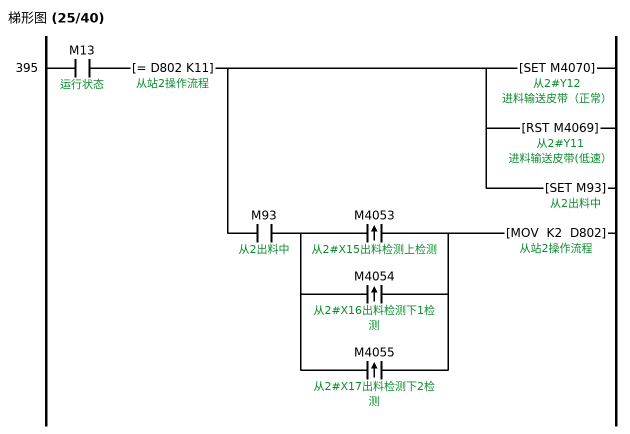
[picture p24: 梯形图 rows 395-395]
LD     M13	; 运行状态
AND=   D802 K11	; 从站2操作流程
SET    M4070	; 从2#Y12 进料输送皮带（正常）
RST    M4069	; 从2#Y11 进料输送皮带(低速）
SET    M93	; 从2出料中
AND    M93	; 从2出料中
LDP    M4053	; 从2#X15出料检测上检测
ORP    M4054	; 从2#X16出料检测下1检测
ORP    M4055	; 从2#X17出料检测下2检测
ANB
MOV    K2 D802	; 从站2操作流程

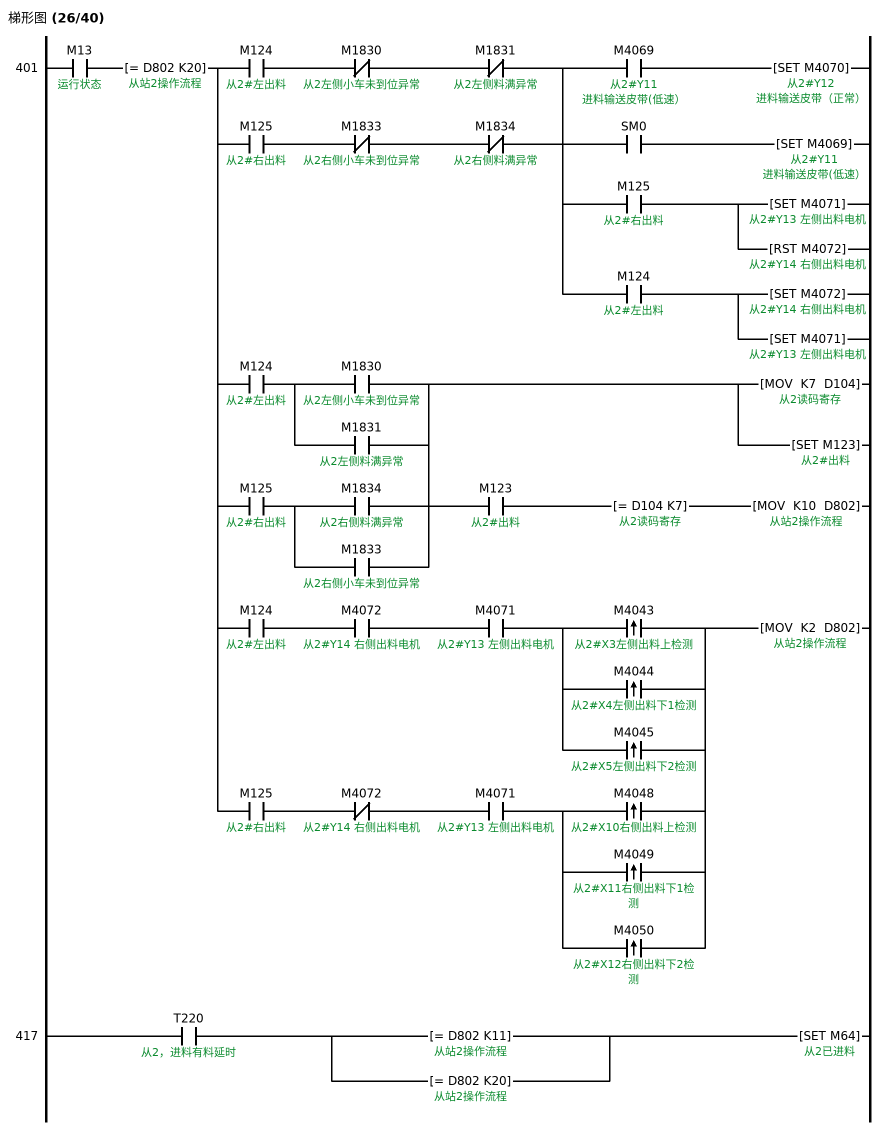
LD     M13	; 运行状态
AND=   D802 K20	; 从站2操作流程
MPS
LD     M124	; 从2#左出料
ANI    M1830	; 从2左侧小车未到位异常
ANI    M1831	; 从2左侧料满异常
LD     M125	; 从2#右出料
ANI    M1833	; 从2右侧小车未到位异常
ANI    M1834	; 从2右侧料满异常
ORB
ANB
MPS
AND    M4069	; 从2#Y11 进料输送皮带(低速）
SET    M4070	; 从2#Y12 进料输送皮带（正常）
MRD
AND    SM0
SET    M4069	; 从2#Y11 进料输送皮带(低速）
MRD
AND    M125	; 从2#右出料
SET    M4071	; 从2#Y13 左侧出料电机
RST    M4072	; 从2#Y14 右侧出料电机
MPP
AND    M124	; 从2#左出料
SET    M4072	; 从2#Y14 右侧出料电机
SET    M4071	; 从2#Y13 左侧出料电机
MRD
LD     M124	; 从2#左出料
LD     M1830	; 从2左侧小车未到位异常
OR     M1831	; 从2左侧料满异常
ANB
LD     M125	; 从2#右出料
LD     M1834	; 从2右侧料满异常
OR     M1833	; 从2右侧小车未到位异常
ANB
ORB
ANB
MOV    K7 D104	; 从2读码寄存
SET    M123	; 从2#出料
AND    M123	; 从2#出料
AND=   D104 K7	; 从2读码寄存
MOV    K10 D802	; 从站2操作流程
MPP
LD     M124	; 从2#左出料
AND    M4072	; 从2#Y14 右侧出料电机
AND    M4071	; 从2#Y13 左侧出料电机
LDP    M4043	; 从2#X3左侧出料上检测
ORP    M4044	; 从2#X4左侧出料下1检测
ORP    M4045	; 从2#X5左侧出料下2检测
ANB
LD     M125	; 从2#右出料
ANI    M4072	; 从2#Y14 右侧出料电机
AND    M4071	; 从2#Y13 左侧出料电机
LDP    M4048	; 从2#X10右侧出料上检测
ORP    M4049	; 从2#X11右侧出料下1检测
ORP    M4050	; 从2#X12右侧出料下2检测
ANB
ORB
ANB
MOV    K2 D802	; 从站2操作流程
LD     T220	; 从2，进料有料延时
LD=    D802 K11	; 从站2操作流程
OR=    D802 K20	; 从站2操作流程
ANB
SET    M64	; 从2已进料

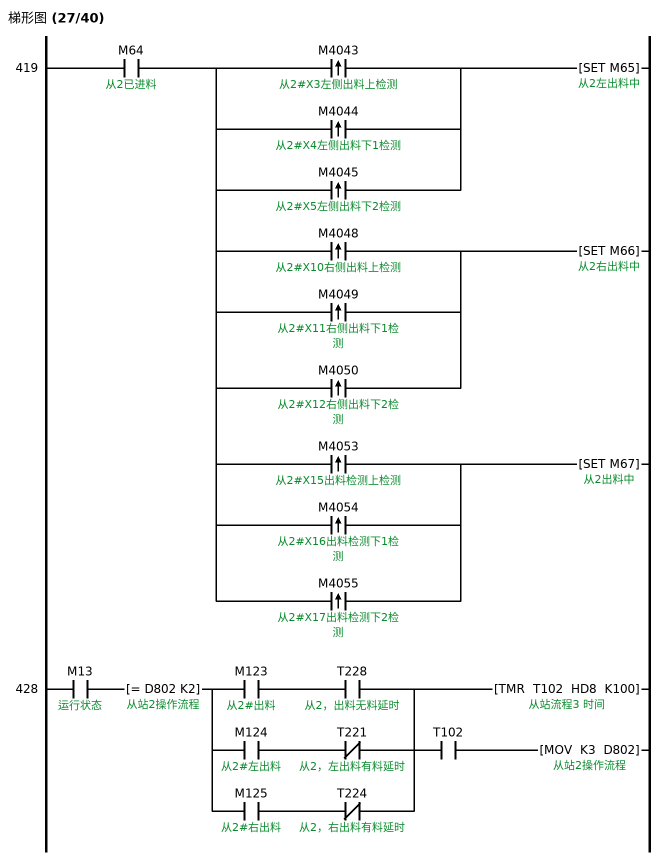
LD     M64	; 从2已进料
MPS
LDP    M4043	; 从2#X3左侧出料上检测
ORP    M4044	; 从2#X4左侧出料下1检测
ORP    M4045	; 从2#X5左侧出料下2检测
ANB
SET    M65	; 从2左出料中
MRD
LDP    M4048	; 从2#X10右侧出料上检测
ORP    M4049	; 从2#X11右侧出料下1检测
ORP    M4050	; 从2#X12右侧出料下2检测
ANB
SET    M66	; 从2右出料中
MPP
LDP    M4053	; 从2#X15出料检测上检测
ORP    M4054	; 从2#X16出料检测下1检测
ORP    M4055	; 从2#X17出料检测下2检测
ANB
SET    M67	; 从2出料中
LD     M13	; 运行状态
AND=   D802 K2	; 从站2操作流程
LD     M123	; 从2#出料
AND    T228	; 从2，出料无料延时
LD     M124	; 从2#左出料
ANI    T221	; 从2，左出料有料延时
ORB
LD     M125	; 从2#右出料
ANI    T224	; 从2，右出料有料延时
ORB
ANB
TMR    T102 HD8 K100	; 从站流程3 时间
AND    T102
MOV    K3 D802	; 从站2操作流程

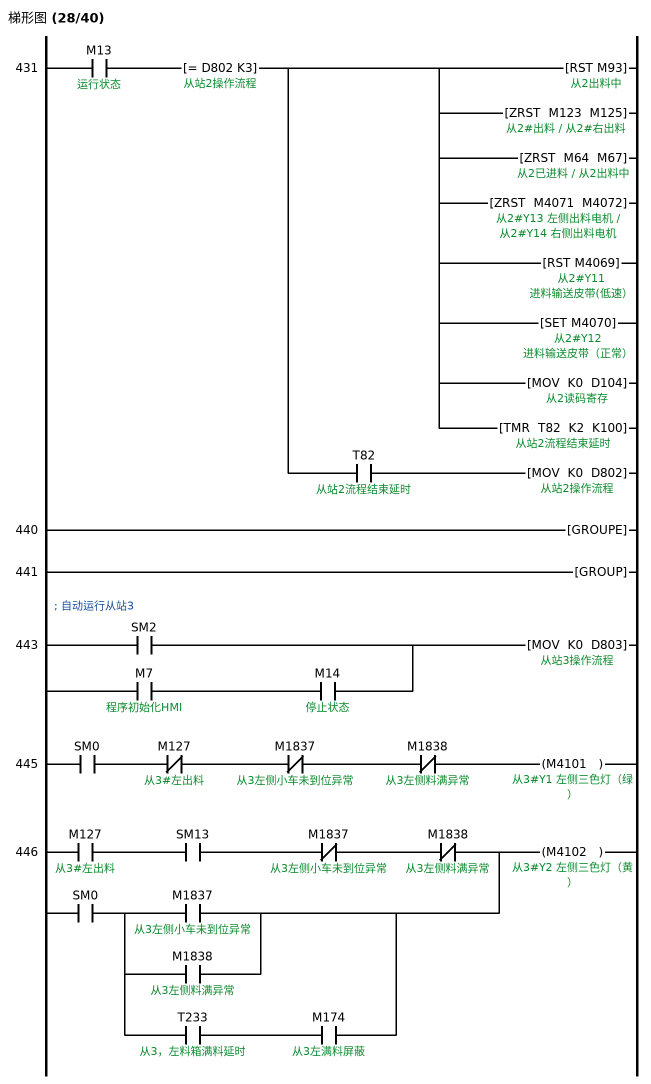
LD     M13	; 运行状态
AND=   D802 K3	; 从站2操作流程
RST    M93	; 从2出料中
ZRST   M123 M125	; 从2#出料 / 从2#右出料
ZRST   M64 M67	; 从2已进料 / 从2出料中
ZRST   M4071 M4072	; 从2#Y13 左侧出料电机 / 从2#Y14 右侧出料电机
RST    M4069	; 从2#Y11 进料输送皮带(低速）
SET    M4070	; 从2#Y12 进料输送皮带（正常）
MOV    K0 D104	; 从2读码寄存
TMR    T82 K2 K100	; 从站2流程结束延时
AND    T82	; 从站2流程结束延时
MOV    K0 D802	; 从站2操作流程
GROUPE
GROUP
; 自动运行从站3
LD     SM2
LD     M7	; 程序初始化HMI
AND    M14	; 停止状态
ORB
MOV    K0 D803	; 从站3操作流程
LD     SM0
ANI    M127	; 从3#左出料
ANI    M1837	; 从3左侧小车未到位异常
ANI    M1838	; 从3左侧料满异常
OUT    M4101	; 从3#Y1 左侧三色灯（绿）
LD     M127	; 从3#左出料
AND    SM13
ANI    M1837	; 从3左侧小车未到位异常
ANI    M1838	; 从3左侧料满异常
LD     SM0
LD     M1837	; 从3左侧小车未到位异常
OR     M1838	; 从3左侧料满异常
LD     T233	; 从3，左料箱满料延时
AND    M174	; 从3左满料屏蔽
ORB
ANB
ORB
OUT    M4102	; 从3#Y2 左侧三色灯（黄）

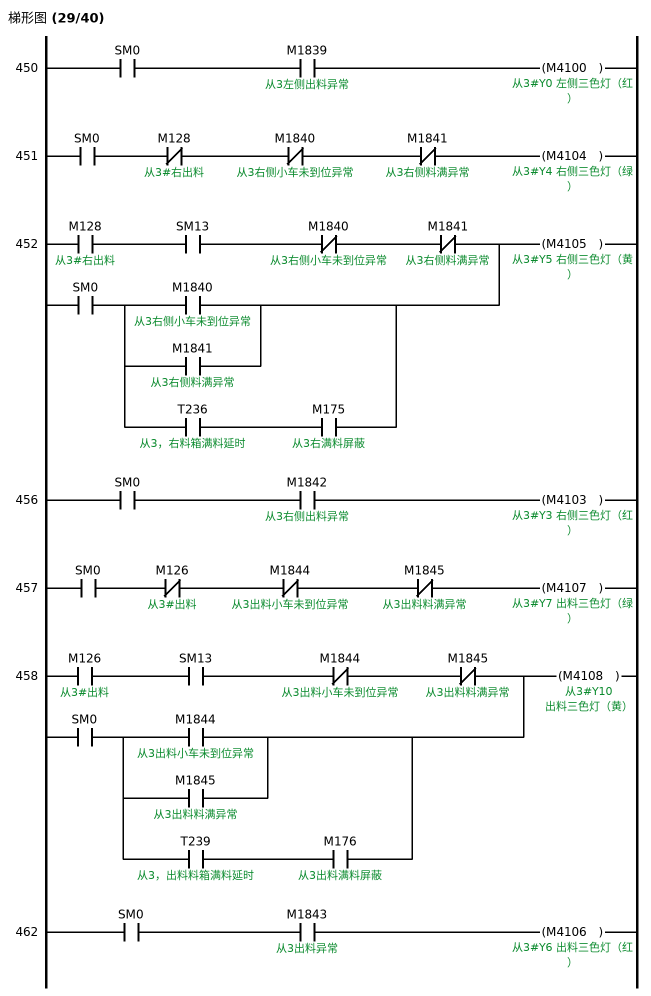
LD     SM0
AND    M1839	; 从3左侧出料异常
OUT    M4100	; 从3#Y0 左侧三色灯（红）
LD     SM0
ANI    M128	; 从3#右出料
ANI    M1840	; 从3右侧小车未到位异常
ANI    M1841	; 从3右侧料满异常
OUT    M4104	; 从3#Y4 右侧三色灯（绿）
LD     M128	; 从3#右出料
AND    SM13
ANI    M1840	; 从3右侧小车未到位异常
ANI    M1841	; 从3右侧料满异常
LD     SM0
LD     M1840	; 从3右侧小车未到位异常
OR     M1841	; 从3右侧料满异常
LD     T236	; 从3，右料箱满料延时
AND    M175	; 从3右满料屏蔽
ORB
ANB
ORB
OUT    M4105	; 从3#Y5 右侧三色灯（黄）
LD     SM0
AND    M1842	; 从3右侧出料异常
OUT    M4103	; 从3#Y3 右侧三色灯（红）
LD     SM0
ANI    M126	; 从3#出料
ANI    M1844	; 从3出料小车未到位异常
ANI    M1845	; 从3出料料满异常
OUT    M4107	; 从3#Y7 出料三色灯（绿）
LD     M126	; 从3#出料
AND    SM13
ANI    M1844	; 从3出料小车未到位异常
ANI    M1845	; 从3出料料满异常
LD     SM0
LD     M1844	; 从3出料小车未到位异常
OR     M1845	; 从3出料料满异常
LD     T239	; 从3，出料料箱满料延时
AND    M176	; 从3出料满料屏蔽
ORB
ANB
ORB
OUT    M4108	; 从3#Y10 出料三色灯（黄）
LD     SM0
AND    M1843	; 从3出料异常
OUT    M4106	; 从3#Y6 出料三色灯（红）

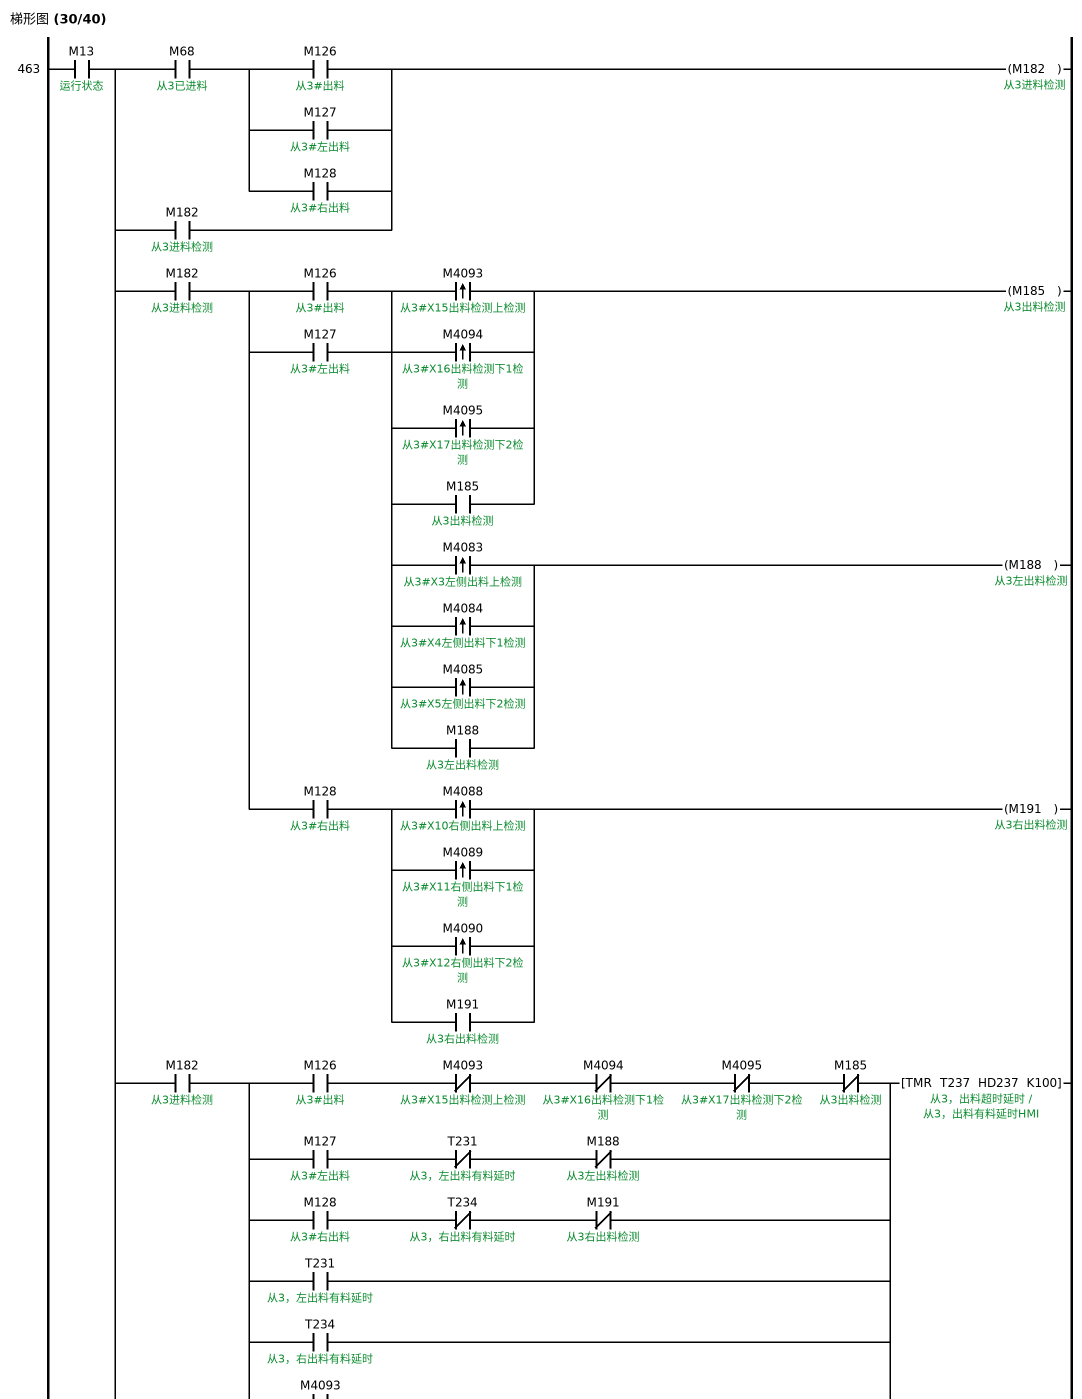
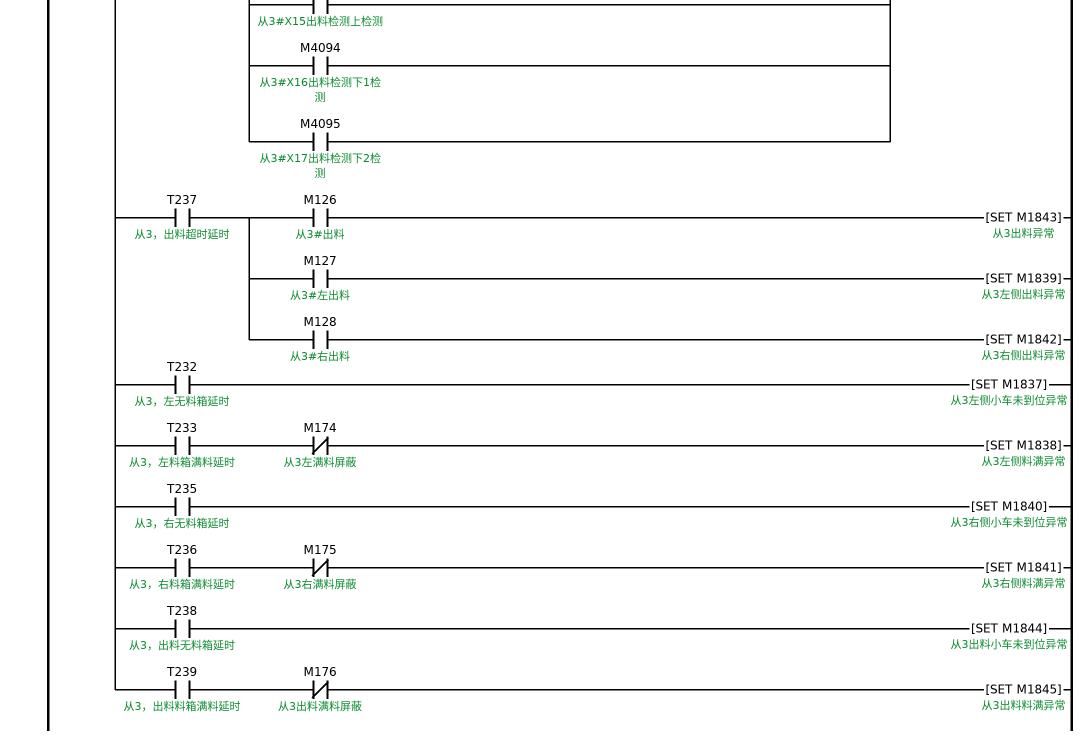
LD     M13	; 运行状态
MPS
LD     M68	; 从3已进料
LD     M126	; 从3#出料
OR     M127	; 从3#左出料
OR     M128	; 从3#右出料
ANB
OR     M182	; 从3进料检测
ANB
OUT    M182	; 从3进料检测
MRD
AND    M182	; 从3进料检测
MPS
LD     M126	; 从3#出料
OR     M127	; 从3#左出料
ANB
MPS
LDP    M4093	; 从3#X15出料检测上检测
ORP    M4094	; 从3#X16出料检测下1检测
ORP    M4095	; 从3#X17出料检测下2检测
OR     M185	; 从3出料检测
ANB
OUT    M185	; 从3出料检测
MPP
LDP    M4083	; 从3#X3左侧出料上检测
ORP    M4084	; 从3#X4左侧出料下1检测
ORP    M4085	; 从3#X5左侧出料下2检测
OR     M188	; 从3左出料检测
ANB
OUT    M188	; 从3左出料检测
MPP
AND    M128	; 从3#右出料
LDP    M4088	; 从3#X10右侧出料上检测
ORP    M4089	; 从3#X11右侧出料下1检测
ORP    M4090	; 从3#X12右侧出料下2检测
OR     M191	; 从3右出料检测
ANB
OUT    M191	; 从3右出料检测
MRD
AND    M182	; 从3进料检测
LD     M126	; 从3#出料
ANI    M4093	; 从3#X15出料检测上检测
ANI    M4094	; 从3#X16出料检测下1检测
ANI    M4095	; 从3#X17出料检测下2检测
ANI    M185	; 从3出料检测
LD     M127	; 从3#左出料
ANI    T231	; 从3，左出料有料延时
ANI    M188	; 从3左出料检测
ORB
LD     M128	; 从3#右出料
ANI    T234	; 从3，右出料有料延时
ANI    M191	; 从3右出料检测
ORB
OR     T231	; 从3，左出料有料延时
OR     T234	; 从3，右出料有料延时
OR     M4093	; 从3#X15出料检测上检测
OR     M4094	; 从3#X16出料检测下1检测
OR     M4095	; 从3#X17出料检测下2检测
ANB
TMR    T237 HD237 K100	; 从3，出料超时延时 / 从3，出料有料延时HMI
MRD
AND    T237	; 从3，出料超时延时
MPS
AND    M126	; 从3#出料
SET    M1843	; 从3出料异常
MRD
AND    M127	; 从3#左出料
SET    M1839	; 从3左侧出料异常
MPP
AND    M128	; 从3#右出料
SET    M1842	; 从3右侧出料异常
MRD
AND    T232	; 从3，左无料箱延时
SET    M1837	; 从3左侧小车未到位异常
MRD
AND    T233	; 从3，左料箱满料延时
ANI    M174	; 从3左满料屏蔽
SET    M1838	; 从3左侧料满异常
MRD
AND    T235	; 从3，右无料箱延时
SET    M1840	; 从3右侧小车未到位异常
MRD
AND    T236	; 从3，右料箱满料延时
ANI    M175	; 从3右满料屏蔽
SET    M1841	; 从3右侧料满异常
MRD
AND    T238	; 从3，出料无料箱延时
SET    M1844	; 从3出料小车未到位异常
MPP
AND    T239	; 从3，出料料箱满料延时
ANI    M176	; 从3出料满料屏蔽
SET    M1845	; 从3出料料满异常

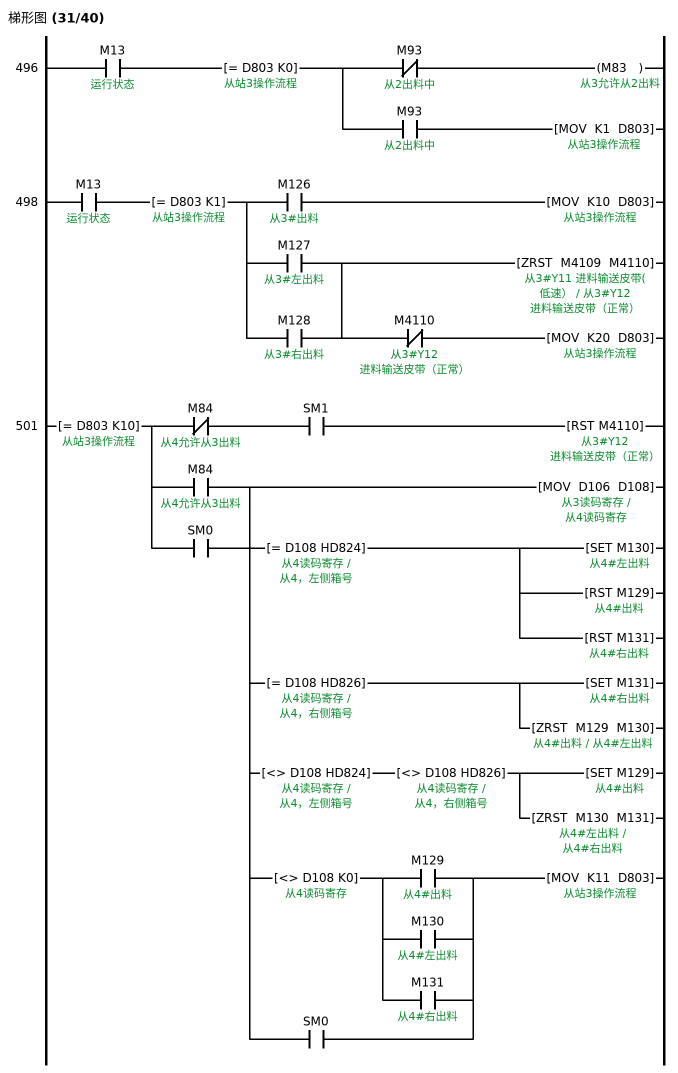
LD     M13	; 运行状态
AND=   D803 K0	; 从站3操作流程
MPS
ANI    M93	; 从2出料中
OUT    M83	; 从3允许从2出料
MPP
AND    M93	; 从2出料中
MOV    K1 D803	; 从站3操作流程
LD     M13	; 运行状态
AND=   D803 K1	; 从站3操作流程
MPS
AND    M126	; 从3#出料
MOV    K10 D803	; 从站3操作流程
MPP
LD     M127	; 从3#左出料
OR     M128	; 从3#右出料
ANB
ZRST   M4109 M4110	; 从3#Y11 进料输送皮带(低速） / 从3#Y12 进料输送皮带（正常）
ANI    M4110	; 从3#Y12 进料输送皮带（正常）
MOV    K20 D803	; 从站3操作流程
LD=    D803 K10	; 从站3操作流程
MPS
ANI    M84	; 从4允许从3出料
AND    SM1
RST    M4110	; 从3#Y12 进料输送皮带（正常）
MPP
LD     M84	; 从4允许从3出料
OR     SM0
ANB
MOV    D106 D108	; 从3读码寄存 / 从4读码寄存
MPS
AND=   D108 HD824	; 从4读码寄存 / 从4，左侧箱号
SET    M130	; 从4#左出料
RST    M129	; 从4#出料
RST    M131	; 从4#右出料
MRD
AND=   D108 HD826	; 从4读码寄存 / 从4，右侧箱号
SET    M131	; 从4#右出料
ZRST   M129 M130	; 从4#出料 / 从4#左出料
MRD
AND<>  D108 HD824	; 从4读码寄存 / 从4，左侧箱号
AND<>  D108 HD826	; 从4读码寄存 / 从4，右侧箱号
SET    M129	; 从4#出料
ZRST   M130 M131	; 从4#左出料 / 从4#右出料
MPP
LD<>   D108 K0	; 从4读码寄存
LD     M129	; 从4#出料
OR     M130	; 从4#左出料
OR     M131	; 从4#右出料
ANB
OR     SM0
ANB
MOV    K11 D803	; 从站3操作流程

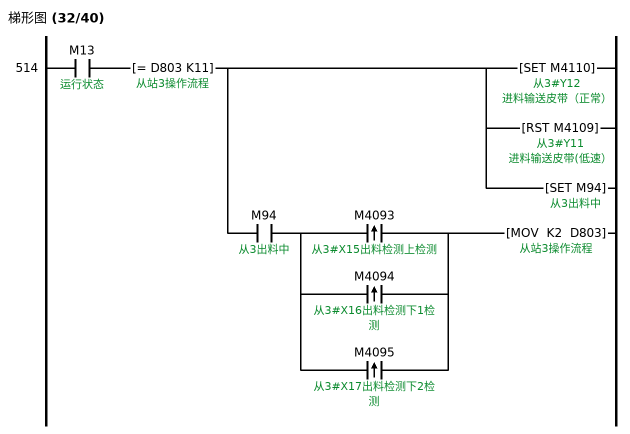
LD     M13	; 运行状态
AND=   D803 K11	; 从站3操作流程
SET    M4110	; 从3#Y12 进料输送皮带（正常）
RST    M4109	; 从3#Y11 进料输送皮带(低速）
SET    M94	; 从3出料中
AND    M94	; 从3出料中
LDP    M4093	; 从3#X15出料检测上检测
ORP    M4094	; 从3#X16出料检测下1检测
ORP    M4095	; 从3#X17出料检测下2检测
ANB
MOV    K2 D803	; 从站3操作流程

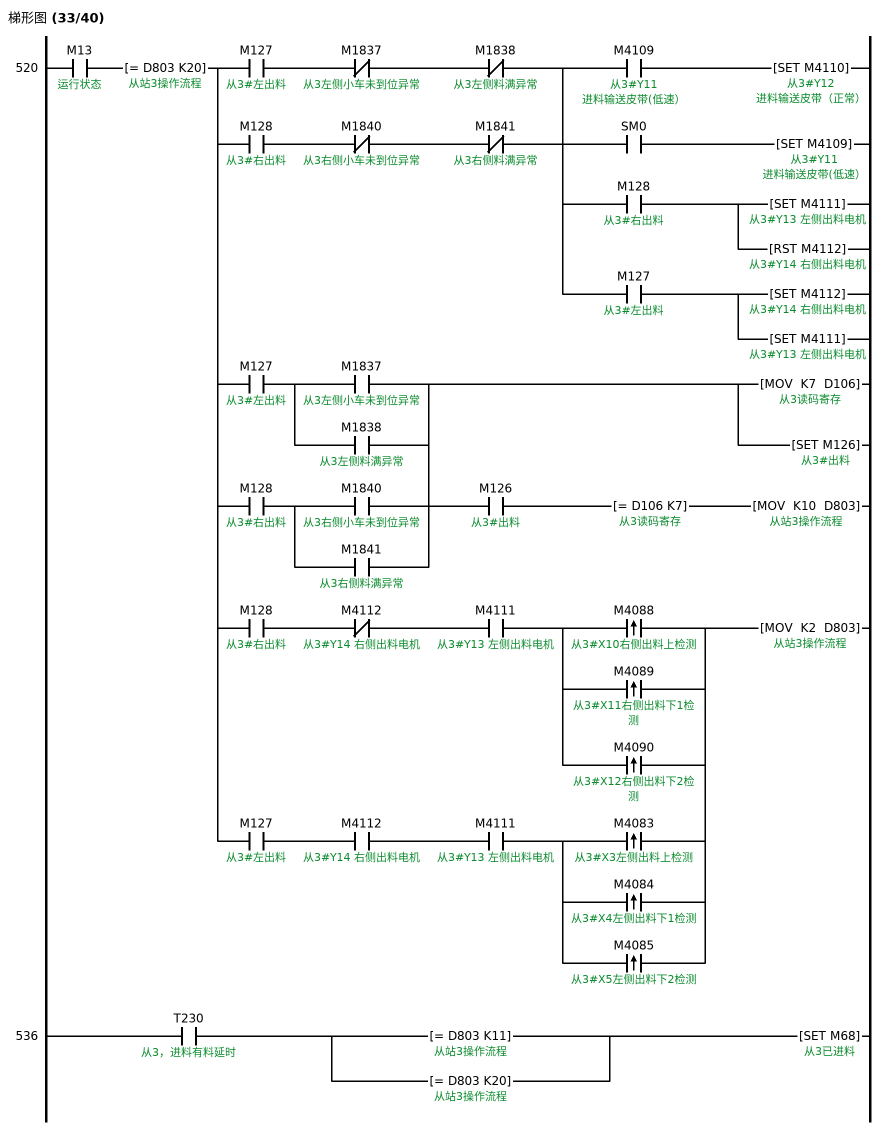
LD     M13	; 运行状态
AND=   D803 K20	; 从站3操作流程
MPS
LD     M127	; 从3#左出料
ANI    M1837	; 从3左侧小车未到位异常
ANI    M1838	; 从3左侧料满异常
LD     M128	; 从3#右出料
ANI    M1840	; 从3右侧小车未到位异常
ANI    M1841	; 从3右侧料满异常
ORB
ANB
MPS
AND    M4109	; 从3#Y11 进料输送皮带(低速）
SET    M4110	; 从3#Y12 进料输送皮带（正常）
MRD
AND    SM0
SET    M4109	; 从3#Y11 进料输送皮带(低速）
MRD
AND    M128	; 从3#右出料
SET    M4111	; 从3#Y13 左侧出料电机
RST    M4112	; 从3#Y14 右侧出料电机
MPP
AND    M127	; 从3#左出料
SET    M4112	; 从3#Y14 右侧出料电机
SET    M4111	; 从3#Y13 左侧出料电机
MRD
LD     M127	; 从3#左出料
LD     M1837	; 从3左侧小车未到位异常
OR     M1838	; 从3左侧料满异常
ANB
LD     M128	; 从3#右出料
LD     M1840	; 从3右侧小车未到位异常
OR     M1841	; 从3右侧料满异常
ANB
ORB
ANB
MOV    K7 D106	; 从3读码寄存
SET    M126	; 从3#出料
AND    M126	; 从3#出料
AND=   D106 K7	; 从3读码寄存
MOV    K10 D803	; 从站3操作流程
MPP
LD     M128	; 从3#右出料
ANI    M4112	; 从3#Y14 右侧出料电机
AND    M4111	; 从3#Y13 左侧出料电机
LDP    M4088	; 从3#X10右侧出料上检测
ORP    M4089	; 从3#X11右侧出料下1检测
ORP    M4090	; 从3#X12右侧出料下2检测
ANB
LD     M127	; 从3#左出料
AND    M4112	; 从3#Y14 右侧出料电机
AND    M4111	; 从3#Y13 左侧出料电机
LDP    M4083	; 从3#X3左侧出料上检测
ORP    M4084	; 从3#X4左侧出料下1检测
ORP    M4085	; 从3#X5左侧出料下2检测
ANB
ORB
ANB
MOV    K2 D803	; 从站3操作流程
LD     T230	; 从3，进料有料延时
LD=    D803 K11	; 从站3操作流程
OR=    D803 K20	; 从站3操作流程
ANB
SET    M68	; 从3已进料

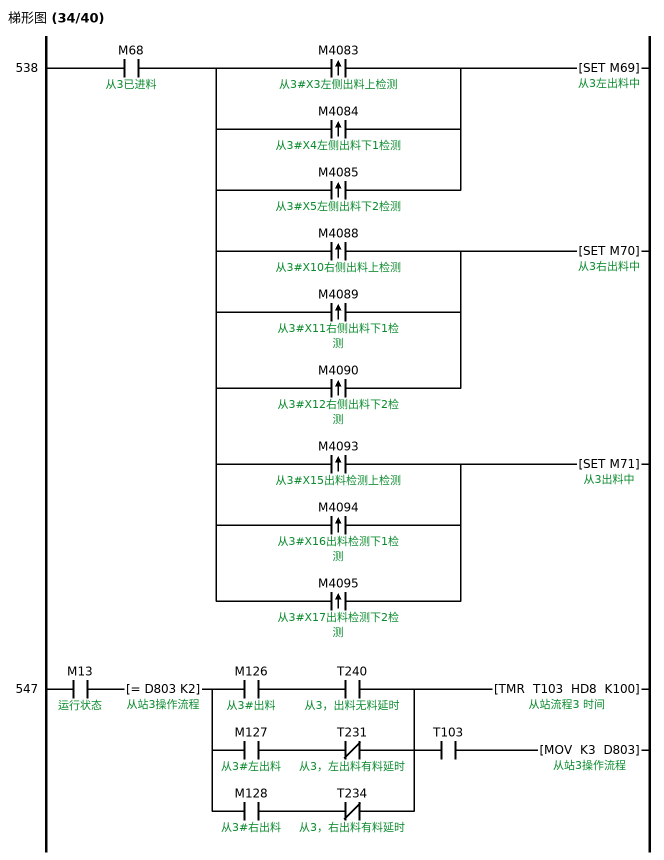
LD     M68	; 从3已进料
MPS
LDP    M4083	; 从3#X3左侧出料上检测
ORP    M4084	; 从3#X4左侧出料下1检测
ORP    M4085	; 从3#X5左侧出料下2检测
ANB
SET    M69	; 从3左出料中
MRD
LDP    M4088	; 从3#X10右侧出料上检测
ORP    M4089	; 从3#X11右侧出料下1检测
ORP    M4090	; 从3#X12右侧出料下2检测
ANB
SET    M70	; 从3右出料中
MPP
LDP    M4093	; 从3#X15出料检测上检测
ORP    M4094	; 从3#X16出料检测下1检测
ORP    M4095	; 从3#X17出料检测下2检测
ANB
SET    M71	; 从3出料中
LD     M13	; 运行状态
AND=   D803 K2	; 从站3操作流程
LD     M126	; 从3#出料
AND    T240	; 从3，出料无料延时
LD     M127	; 从3#左出料
ANI    T231	; 从3，左出料有料延时
ORB
LD     M128	; 从3#右出料
ANI    T234	; 从3，右出料有料延时
ORB
ANB
TMR    T103 HD8 K100	; 从站流程3 时间
AND    T103
MOV    K3 D803	; 从站3操作流程

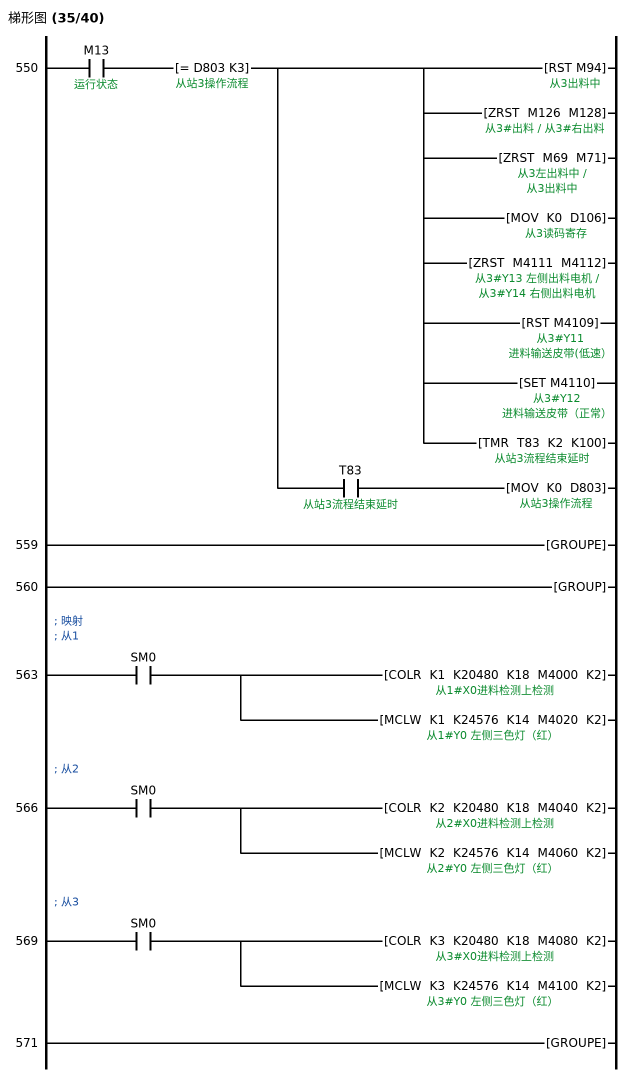
LD     M13	; 运行状态
AND=   D803 K3	; 从站3操作流程
RST    M94	; 从3出料中
ZRST   M126 M128	; 从3#出料 / 从3#右出料
ZRST   M69 M71	; 从3左出料中 / 从3出料中
MOV    K0 D106	; 从3读码寄存
ZRST   M4111 M4112	; 从3#Y13 左侧出料电机 / 从3#Y14 右侧出料电机
RST    M4109	; 从3#Y11 进料输送皮带(低速）
SET    M4110	; 从3#Y12 进料输送皮带（正常）
TMR    T83 K2 K100	; 从站3流程结束延时
AND    T83	; 从站3流程结束延时
MOV    K0 D803	; 从站3操作流程
GROUPE
GROUP
; 映射
; 从1
LD     SM0
COLR   K1 K20480 K18 M4000 K2	; 从1#X0进料检测上检测
MCLW   K1 K24576 K14 M4020 K2	; 从1#Y0 左侧三色灯（红）
; 从2
LD     SM0
COLR   K2 K20480 K18 M4040 K2	; 从2#X0进料检测上检测
MCLW   K2 K24576 K14 M4060 K2	; 从2#Y0 左侧三色灯（红）
; 从3
LD     SM0
COLR   K3 K20480 K18 M4080 K2	; 从3#X0进料检测上检测
MCLW   K3 K24576 K14 M4100 K2	; 从3#Y0 左侧三色灯（红）
GROUPE

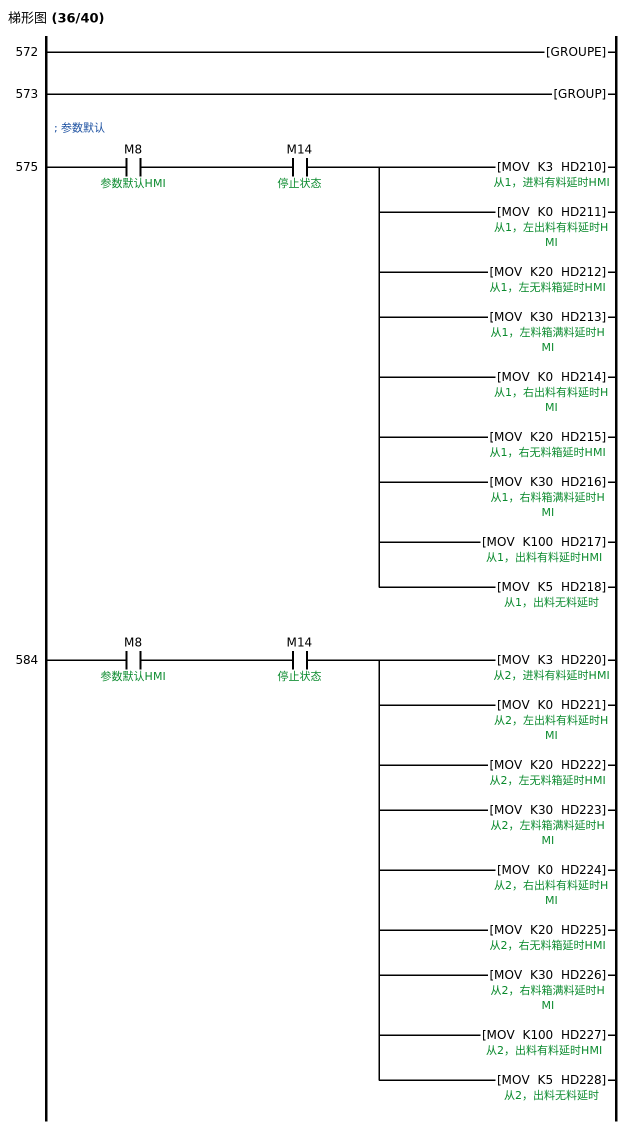
GROUPE
GROUP
; 参数默认
LD     M8	; 参数默认HMI
AND    M14	; 停止状态
MOV    K3 HD210	; 从1，进料有料延时HMI
MOV    K0 HD211	; 从1，左出料有料延时HMI
MOV    K20 HD212	; 从1，左无料箱延时HMI
MOV    K30 HD213	; 从1，左料箱满料延时HMI
MOV    K0 HD214	; 从1，右出料有料延时HMI
MOV    K20 HD215	; 从1，右无料箱延时HMI
MOV    K30 HD216	; 从1，右料箱满料延时HMI
MOV    K100 HD217	; 从1，出料有料延时HMI
MOV    K5 HD218	; 从1，出料无料延时
LD     M8	; 参数默认HMI
AND    M14	; 停止状态
MOV    K3 HD220	; 从2，进料有料延时HMI
MOV    K0 HD221	; 从2，左出料有料延时HMI
MOV    K20 HD222	; 从2，左无料箱延时HMI
MOV    K30 HD223	; 从2，左料箱满料延时HMI
MOV    K0 HD224	; 从2，右出料有料延时HMI
MOV    K20 HD225	; 从2，右无料箱延时HMI
MOV    K30 HD226	; 从2，右料箱满料延时HMI
MOV    K100 HD227	; 从2，出料有料延时HMI
MOV    K5 HD228	; 从2，出料无料延时

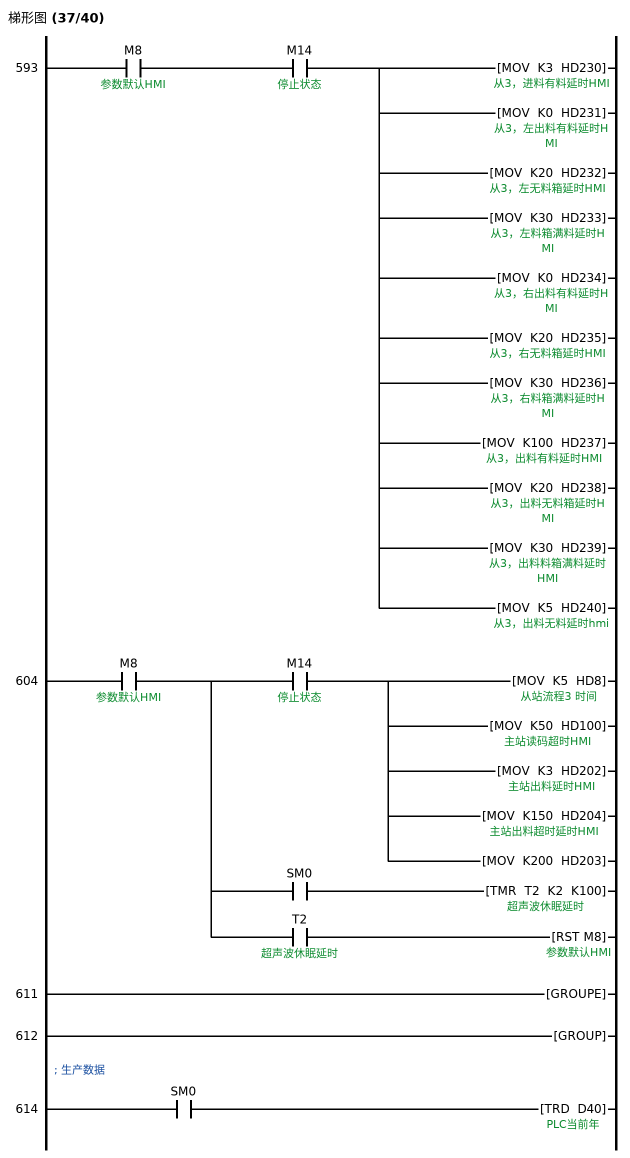
LD     M8	; 参数默认HMI
AND    M14	; 停止状态
MOV    K3 HD230	; 从3，进料有料延时HMI
MOV    K0 HD231	; 从3，左出料有料延时HMI
MOV    K20 HD232	; 从3，左无料箱延时HMI
MOV    K30 HD233	; 从3，左料箱满料延时HMI
MOV    K0 HD234	; 从3，右出料有料延时HMI
MOV    K20 HD235	; 从3，右无料箱延时HMI
MOV    K30 HD236	; 从3，右料箱满料延时HMI
MOV    K100 HD237	; 从3，出料有料延时HMI
MOV    K20 HD238	; 从3，出料无料箱延时HMI
MOV    K30 HD239	; 从3，出料料箱满料延时HMI
MOV    K5 HD240	; 从3，出料无料延时hmi
LD     M8	; 参数默认HMI
MPS
AND    M14	; 停止状态
MOV    K5 HD8	; 从站流程3 时间
MOV    K50 HD100	; 主站读码超时HMI
MOV    K3 HD202	; 主站出料延时HMI
MOV    K150 HD204	; 主站出料超时延时HMI
MOV    K200 HD203
MRD
AND    SM0
TMR    T2 K2 K100	; 超声波休眠延时
MPP
AND    T2	; 超声波休眠延时
RST    M8	; 参数默认HMI
GROUPE
GROUP
; 生产数据
LD     SM0
TRD    D40	; PLC当前年

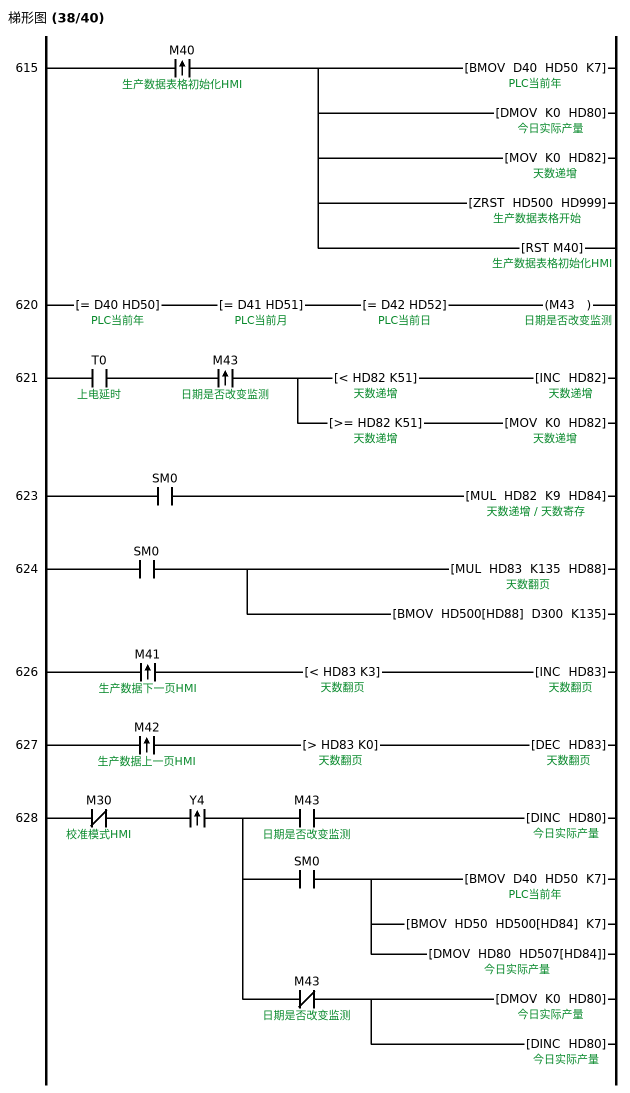
LDP    M40	; 生产数据表格初始化HMI
BMOV   D40 HD50 K7	; PLC当前年
DMOV   K0 HD80	; 今日实际产量
MOV    K0 HD82	; 天数递增
ZRST   HD500 HD999	; 生产数据表格开始
RST    M40	; 生产数据表格初始化HMI
LD=    D40 HD50	; PLC当前年
AND=   D41 HD51	; PLC当前月
AND=   D42 HD52	; PLC当前日
OUT    M43	; 日期是否改变监测
LD     T0	; 上电延时
ANDP   M43	; 日期是否改变监测
MPS
AND<   HD82 K51	; 天数递增
INC    HD82	; 天数递增
MPP
AND>=  HD82 K51	; 天数递增
MOV    K0 HD82	; 天数递增
LD     SM0
MUL    HD82 K9 HD84	; 天数递增 / 天数寄存
LD     SM0
MUL    HD83 K135 HD88	; 天数翻页
BMOV   HD500[HD88] D300 K135
LDP    M41	; 生产数据下一页HMI
AND<   HD83 K3	; 天数翻页
INC    HD83	; 天数翻页
LDP    M42	; 生产数据上一页HMI
AND>   HD83 K0	; 天数翻页
DEC    HD83	; 天数翻页
LDI    M30	; 校准模式HMI
ANDP   Y4
MPS
AND    M43	; 日期是否改变监测
DINC   HD80	; 今日实际产量
MRD
AND    SM0
BMOV   D40 HD50 K7	; PLC当前年
BMOV   HD50 HD500[HD84] K7
DMOV   HD80 HD507[HD84]	; 今日实际产量
MPP
ANI    M43	; 日期是否改变监测
DMOV   K0 HD80	; 今日实际产量
DINC   HD80	; 今日实际产量

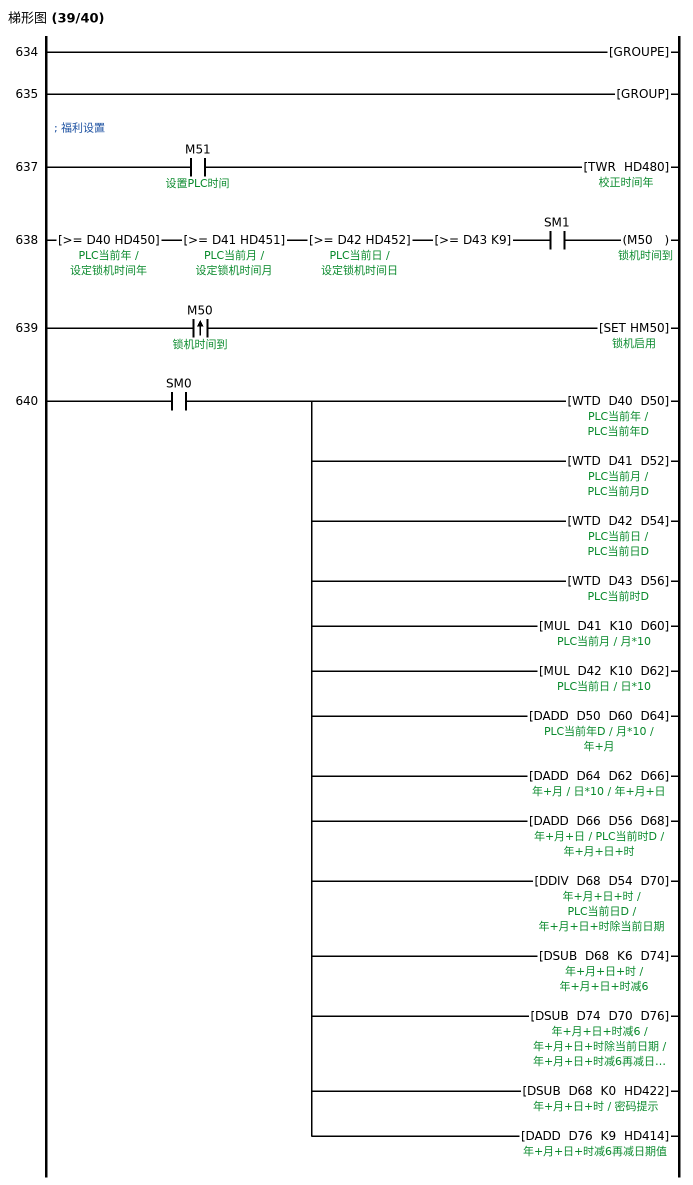
GROUPE
GROUP
; 福利设置
LD     M51	; 设置PLC时间
TWR    HD480	; 校正时间年
LD>=   D40 HD450	; PLC当前年 / 设定锁机时间年
AND>=  D41 HD451	; PLC当前月 / 设定锁机时间月
AND>=  D42 HD452	; PLC当前日 / 设定锁机时间日
AND>=  D43 K9
AND    SM1
OUT    M50	; 锁机时间到
LDP    M50	; 锁机时间到
SET    HM50	; 锁机启用
LD     SM0
WTD    D40 D50	; PLC当前年 / PLC当前年D
WTD    D41 D52	; PLC当前月 / PLC当前月D
WTD    D42 D54	; PLC当前日 / PLC当前日D
WTD    D43 D56	; PLC当前时D
MUL    D41 K10 D60	; PLC当前月 / 月*10
MUL    D42 K10 D62	; PLC当前日 / 日*10
DADD   D50 D60 D64	; PLC当前年D / 月*10 / 年+月
DADD   D64 D62 D66	; 年+月 / 日*10 / 年+月+日
DADD   D66 D56 D68	; 年+月+日 / PLC当前时D / 年+月+日+时
DDIV   D68 D54 D70	; 年+月+日+时 / PLC当前日D / 年+月+日+时除当前日期
DSUB   D68 K6 D74	; 年+月+日+时 / 年+月+日+时减6
DSUB   D74 D70 D76	; 年+月+日+时减6 / 年+月+日+时除当前日期 / 年+月+日+时减6再减日期值
DSUB   D68 K0 HD422	; 年+月+日+时 / 密码提示
DADD   D76 K9 HD414	; 年+月+日+时减6再减日期值

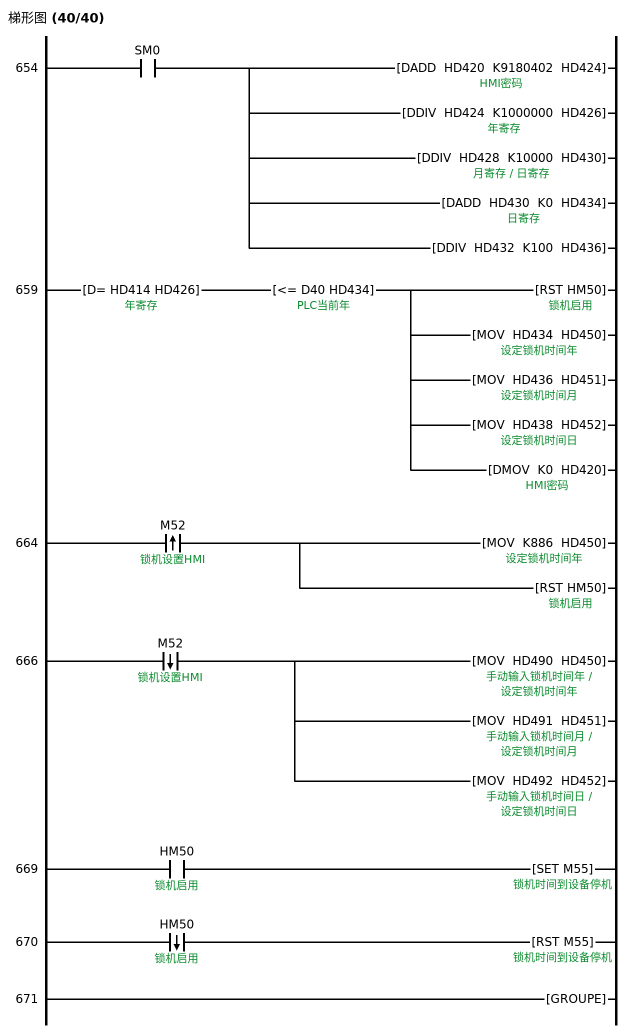
LD     SM0
DADD   HD420 K9180402 HD424	; HMI密码
DDIV   HD424 K1000000 HD426	; 年寄存
DDIV   HD428 K10000 HD430	; 月寄存 / 日寄存
DADD   HD430 K0 HD434	; 日寄存
DDIV   HD432 K100 HD436
DLD=   HD414 HD426	; 年寄存
AND<=  D40 HD434	; PLC当前年
RST    HM50	; 锁机启用
MOV    HD434 HD450	; 设定锁机时间年
MOV    HD436 HD451	; 设定锁机时间月
MOV    HD438 HD452	; 设定锁机时间日
DMOV   K0 HD420	; HMI密码
LDP    M52	; 锁机设置HMI
MOV    K886 HD450	; 设定锁机时间年
RST    HM50	; 锁机启用
LDF    M52	; 锁机设置HMI
MOV    HD490 HD450	; 手动输入锁机时间年 / 设定锁机时间年
MOV    HD491 HD451	; 手动输入锁机时间月 / 设定锁机时间月
MOV    HD492 HD452	; 手动输入锁机时间日 / 设定锁机时间日
LD     HM50	; 锁机启用
SET    M55	; 锁机时间到设备停机
LDF    HM50	; 锁机启用
RST    M55	; 锁机时间到设备停机
GROUPE

COMMENTS (devices not used above)
X15	进料检测下1检测
X16	进料检测下2检测
M3	急停HMI
M5	NG清料HMI
M6	轴复位HMI
M9	产量清零HMI
M10	当前产量清零HMI
M21	軸总復位中
M22	设备复位中
M25	设备清料完成
M2042	轴2_JOG快慢速HMI
M2021	轴1_JOG- HMI
M2022	轴2_JOG- HMI
M2041	轴1_JOG快慢速HMI
M2002	轴2_JOG+ HMI
HD200	主站进料有料延时HMI
D2100	轴1_JOG快速度
D2102	轴1_JOG慢速度
D2104	轴1_JOG速度寄存
D2106	轴1_JOG增量
D2108	轴1_JOG位置寄存
D2110	轴1_回零速度
D2112	轴1_运行速度
D2114	轴1_自动加速度
D2115	轴1_自动减速度
D2116	轴1_JOG加速度
D2117	轴1_JOG减速度
D2118	轴1_定位位置寄存
M2141	轴1_伺服回零中
M1200	快慢速切换HMI
M1020	从1#Y0 左侧三色灯（红）       HMI
HD12	滚刀切料个数计数
M2001	轴1_JOG+ HMI
HD40	Y0当前脉冲值记忆
HD42	Y1当前脉冲值记忆
HD2	超声波休眠时间
T3	超声运行延时
D110	从5读码寄存
D112	从6读码寄存
D114	从7读码寄存
D116	从8读码寄存
D118	从9读码寄存
D120	从10读码寄存
D122	从11读码寄存
D124	从12读码寄存
D126	从13读码寄存
D142	输出脉冲频率浮点数
HD32	生产效率寄存2
HD20	设定产量HMI
HD22	实际产量(切鼻梁个数计数)
HD30	生产效率寄存1
M1600	产量达成
HM30	内置鼻梁标志/外置鼻梁HMI
HD24	滚刀切料个数计数
HD34	生产效率
HM32	校准完成
HM3	急停后切断鼻梁
M18	手动操作记忆标志
HD507	当日实际产量
HD453	设定锁机时间时
HD481	校正时间月
HD482	校正时间日
HD483	校正时间时
D72	年+月+日+时除当前日期得商
HD28	累计产量
HD10	流程结束，电机保持时间
X10000	书本到位感应器1（电机侧斜面）       书本到位感应器1
X10001	书本到位感应器2（斜面）             书本到位感应器2
X10002	书本到位感应器3（斜面）             书本到位感应器3
X10003	小车感应光栅
X10004	小车到位感应（对射）
X10005	防压手感应器
X10006	书枰感应器7
X10007	书本感应器8
M2101	轴1_伺服回零HMI
M2102	轴2_伺服回零HMI
M2121	轴1_伺服回零允许
M2122	轴2_伺服回零允许
M2142	轴2_伺服回零中
M2161	轴1_原点确定
M2162	轴2_原点确定
M2181	轴1_定位允许
M2182	轴2_定位允许
M2201	轴1_JOG连续/增量HMI
M2202	轴2_JOG连续/增量HMI
M2241	轴1_增量JOG运行
M2242	轴2_增量JOG运行
M2310	轴1-伺服原点运行HMI
M2311	轴1-伺服定位运行HMI
M2320	轴2-伺服原点运行HMI
M2321	轴2-伺服定位运行HMI
M2510	轴1-伺服原点运行
M2511	轴1-伺服定位运行
M2520	轴2-伺服原点运行
M2521	轴2-伺服定位运行
M2710	轴1-伺服原点位置
M2711	轴1-伺服定位位置
M2720	轴2-伺服原点位置
M2721	轴2-伺服定位位置
HD832	从5，左侧箱号
HD834	从5，右侧箱号
HD836	从5，出料箱号
HD840	从6，左侧箱号
HD842	从6，右侧箱号
HD844	从6，出料箱号
HD848	从7，左侧箱号
HD850	从7，右侧箱号
HD852	从7，出料箱号
HD856	从8，左侧箱号
HD812	从2，出料箱号
HD804	从1，出料箱号
HD868	从9，出料箱号
HD872	从10，左侧箱号
HD874	从10，右侧箱号
HD876	从10，出料箱号
HD880	从11，左侧箱号
HD882	从11，右侧箱号
HD884	从11，出料箱号
HD888	从12，左侧箱号
HD890	从12，右侧箱号
HD892	从12，出料箱号
HD858	从8，右侧箱号
HD860	从8，出料箱号
HD864	从9，左侧箱号
HD866	从9，右侧箱号
D851	轴1-回原点流程
HD828	从4，出料箱号
T422	轴1 启动
M1021	从1#Y1 左侧三色灯（绿）       HMI
D852	轴2-回原流程
T424	轴2定位允许
M2312	还书位置运行-HMI
M2512	轴1-还书位置运行
M2712	轴1-还书位置
D810	从站10操作流程
D2501	书本识别启动PLC写1，收到完成信号后PLC置0
D2502	PLC写1，书满暂停，处理完后PLC置0
M1022	从1#Y2 左侧三色灯（黄）       HMI
M1023	从1#Y3 右侧三色灯（红）       HMI
M1024	从1#Y4 右侧三色灯（绿）       HMI
M1025	从1#Y5 右侧三色灯（黄）       HMI
M1026	从1#Y6 出料三色灯（红）       HMI
M1027	从1#Y7 出料三色灯（绿）       HMI
M1028	从1#Y10 出料三色灯（黄）       HMI
M1030	从1#Y12 进料输送皮带（正常）       HMI
T201	主站出料有料延时
M1040	从2#Y0 左侧三色灯（红）       HMI
M1041	从2#Y1 左侧三色灯（绿）       HMI
M1042	从2#Y2 左侧三色灯（黄）       HMI
M1043	从2#Y3 右侧三色灯（红）       HMI
M1044	从2#Y4 右侧三色灯（绿）       HMI
M1045	从2#Y5 右侧三色灯（黄）       HMI
M1046	从2#Y6 出料三色灯（红）       HMI
M1047	从2#Y7 出料三色灯（绿）       HMI
M1048	从2#Y10 出料三色灯（黄）       HMI
M1050	从2#Y12 进料输送皮带（正常）       HMI
M1060	从3#Y0 左侧三色灯（红）       HMI
M1061	从3#Y1 左侧三色灯（绿）       HMI
M1062	从3#Y2 左侧三色灯（黄）       HMI
M1063	从3#Y3 右侧三色灯（红）       HMI
M1064	从3#Y4 右侧三色灯（绿）       HMI
M1065	从3#Y5 右侧三色灯（黄）       HMI
M1066	从3#Y6 出料三色灯（红）       HMI
M1067	从3#Y7 出料三色灯（绿）       HMI
M1068	从3#Y10 出料三色灯（黄）       HMI
M1070	从3#Y12 进料输送皮带（正常）       HMI
M4026	从1#Y6 出料三色灯（红）
M4027	从1#Y7 出料三色灯（绿）
M4028	从1#Y10 出料三色灯（黄）
M4066	从2#Y6 出料三色灯（红）
M4067	从2#Y7 出料三色灯（绿）
M4068	从2#Y10 出料三色灯（黄）
HD201	主站出料有料延时HMI
M103	从站4#进料皮带速度切换=0 正常，=1低速
M104	从站5#进料皮带速度切换=0 正常，=1低速
M105	从站6#进料皮带速度切换=0 正常，=1低速
M106	从站7#进料皮带速度切换=0 正常，=1低速
M107	从站8#进料皮带速度切换=0 正常，=1低速
M108	从站9#进料皮带速度切换=0 正常，=1低速
M109	从站10#进料皮带速度切换=0 正常，=1低速
M110	从站11#进料皮带速度切换=0 正常，=1低速
M111	从站12#进料皮带速度切换=0 正常，=1低速
M112	从站13#进料皮带速度切换=0 正常，=1低速
M1610	主站已进料
T401	主站出料超时
M1611	从1已进料
M132	从5#出料
M133	从5#左出料
M134	从5#右出料
M135	从6#出料
M136	从6#左出料
M137	从6#右出料
M138	从7#出料
M139	从7#左出料
M140	从7#右出料
M141	从8#出料
M142	从8#左出料
M143	从8#右出料
M144	从9#出料
M145	从9#左出料
M146	从9#右出料
M147	从10#出料
M148	从10#左出料
M149	从10#右出料
M150	从11#出料
M151	从11#左出料
M152	从11#右出料
M153	从12#出料
M154	从12#左出料
M155	从12#右出料
M156	从13#出料
M157	从13#左出料
D804	从站4操作流程
D805	从站5操作流程
D806	从站6操作流程
D807	从站7操作流程
D808	从站8操作流程
D809	从站9操作流程
D811	从站11操作流程
D812	从站12操作流程
D813	从站13操作流程
T80	主站流程结束延时
T84	从站4流程结束延时
T85	从站5流程结束延时
T86	从站6流程结束延时
T87	从站7流程结束延时
T88	从站8流程结束延时
T89	从站9流程结束延时
T90	从站10流程结束延时
T91	从站11流程结束延时
T92	从站12流程结束延时
T93	从站13流程结束延时
T219	从1流程结束，电机保持时间
T229	从2流程结束，电机保持时间
T241	从3流程结束，电机保持时间
HD219	从1流程结束，电机保持时间HMI
HD229	从2流程结束，电机保持时间HMI